// TIA Portal project "TestwithPSC" (V20)

(* hardware
DEVICE "S7-1500/ET200MP station_1"  S7-1500 station
   slot 0: "Rail_0"  Rack  6ES7 590-1***0-0AA0
   slot 1: "PLC_1"  CPU 1516F-3 PN/DP  6ES7 516-3FN01-0AB0  V2.9
      slot 3: "CPU display_1"  6ES7591-1BA00-0AA0
      slot 32768: "PROFINET interface_1"  X1
      slot 33024: "PROFINET interface_2"  X2
      slot 33280: "DP interface_1"  X3
      slot 34817: "Virtual CP interface port_1"  Virtual CP interface port  Virtual CP interface port
DEVICE "GSD device_1"  GSD.Device.PN
   slot 0: "Rack"  Rack  V1.0
   slot 0: "PSC1-C-xxx-FB1-PNPS"  PSC1-C-xxx RE/PNS V3.5.35 - V3.5.x  0000.000  V1.5
      slot 0: "PSC1-C-xxx RE/PNS V3.5.35 - V3.5.x"  PSC1-C-xxx RE/PNS V3.5.35 - V3.5.x
      slot 1: "PN-IO"  PN-IO
         slot 1: "Port 1"  Port 1
         slot 2: "Port 2"  Port 2
   slot 1: "Device Diagnosis_1"  Device Diagnosis
      slot 0: "128 Bytes Input"  128 Bytes Input
   slot 2: "Outputs_1"  Outputs
      slot 0: "4 Bytes Output"  4 Bytes Output
   slot 3: "SD Bus Input_1"  SD Bus Input
      slot 0: "64 Bytes Input"  64 Bytes Input
   slot 4: "SD Bus Output_1"  SD Bus Output
      slot 0: "64 Bytes Output"  64 Bytes Output
   slot 5: "F-Module I/O (12 Bytes)_1"  F-Module I/O (12 Bytes)
      slot 0: "F-Module I/O (12 Bytes)"  F-Module I/O (12 Bytes)
*)

// ===== PLC "PLC_1"  CPU 1516F-3 PN/DP =====

VAR_GLOBAL   // PLC tag table "Default tag table"
   "mReset" AT %M30.0 : Bool;
   "mReset1" AT %M3.1 : Bool;
   "mNetworkResetCmd" AT %M3.2 : Bool;
   "SafetyResetNetworkCmd" AT %Q200.0 : Bool;
   "SafetyINLightCurtain" AT %I200.0 : Bool;
END_VAR

VAR_GLOBAL   // PLC tag table "Tag table_1"
   "PSC1_RawData_IN" AT %I0.0 : "udt_128Bytes";
   "PSC1_RawData_OUT" AT %Q0.0 : "udt_4Bytes";
END_VAR

TYPE "udt_PSC_IN"
   STRUCT
      PSCMode : UInt;
      AliveCounter : UInt;
      DeviceError : UInt;
      ErrorCode : UInt;
      LogicData : Array[0..407] of Bool;
   END_STRUCT;
END_TYPE

TYPE "udt_PSC_OUT"
   STRUCT
      LogicData : Array[0..31] of Bool;
   END_STRUCT;
END_TYPE

TYPE "udt_128Bytes"
   STRUCT
      _raw : Array[0..127] of Byte;
   END_STRUCT;
END_TYPE

TYPE "udt_PSC"
   STRUCT
      in : "udt_PSC_IN";
      out : "udt_PSC_OUT";
   END_STRUCT;
END_TYPE

TYPE "udt_4Bytes"
   STRUCT
      _raw : Array[0..3] of Byte;
   END_STRUCT;
END_TYPE

DATA_BLOCK "Main_Safety_RTG1_DB"   // DB1, F_DB
{ S7_Optimized_Access := 'TRUE' }
NAME : FUSI
VERSION : 0.1
// stored: InstanceOfName Main_Safety_RTG1
"Main_Safety_RTG1"
BEGIN
END_DATA_BLOCK

DATA_BLOCK "FB_PSC_DB"   // DB2
{ S7_Optimized_Access := 'TRUE' }
VERSION : 0.1
// stored: InstanceOfName FB_PSC
"FB_PSC"
BEGIN
END_DATA_BLOCK

DATA_BLOCK "DB_PSC"   // DB3
{ S7_Optimized_Access := 'TRUE' }
VERSION : 0.1
BEGIN
END_DATA_BLOCK

DATA_BLOCK "FB_Station_DB"   // DB4
{ S7_Optimized_Access := 'TRUE' }
VERSION : 0.1
// stored: InstanceOfName FB_Station
"FB_Station"
BEGIN
END_DATA_BLOCK

FUNCTION_BLOCK "Main_Safety_RTG1"   // FB1, F_FBD
{ S7_Optimized_Access := 'TRUE' }
   VAR
      ACK_GL_Instance : ACK_GL;
   END_VAR
   VAR_TEMP
      LightCurtainOK : Bool;
   END_VAR
BEGIN

REGION Network 1
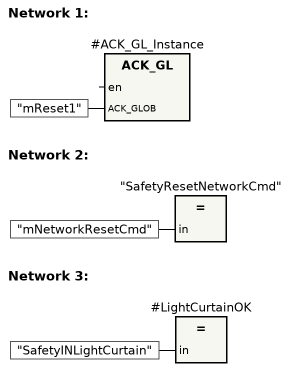
   #ACK_GL_Instance(ACK_GLOB := "mReset1");   // ACK_GL
END_REGION

REGION Network 2
   "SafetyResetNetworkCmd" := "mNetworkResetCmd";
END_REGION

REGION Network 3
   #LightCurtainOK := "SafetyINLightCurtain";
END_REGION
END_FUNCTION_BLOCK

FUNCTION_BLOCK "FB_PSC"   // FB2, LAD
{ S7_Optimized_Access := 'TRUE' }
VERSION : 0.1
   VAR_IN_OUT
      ioRawinputData : Array[*] of Byte;
      ioRawOutputData : Array[*] of Byte;
      ioData : "udt_PSC";
   END_VAR
   VAR_TEMP
      iCounter : Int;
      iIndex : Int;
   END_VAR
BEGIN

REGION Network 2 (SCL)
   #iIndex := 0;
   FOR #iCounter := 5 TO 55 DO

       #ioData.in.LogicData[#iIndex*8]:=
       #ioRawinputData[#iCounter].%X0;

       #ioData.in.LogicData[#iIndex*8+1] :=
       #ioRawinputData[#iCounter].%X1;

       #ioData.in.LogicData[#iIndex*8+2] :=
       #ioRawinputData[#iCounter].%X2;

       #ioData.in.LogicData[#iIndex * 8 + 3] :=
       #ioRawinputData[#iCounter].%X3;

       #ioData.in.LogicData[#iIndex*8+4] :=
       #ioRawinputData[#iCounter].%X4;

       #ioData.in.LogicData[#iIndex * 8 + 5] :=
       #ioRawinputData[#iCounter].%X5;

       #ioData.in.LogicData[#iIndex * 8 + 6] :=
       #ioRawinputData[#iCounter].%X6;

       #ioData.in.LogicData[#iIndex * 8 + 7] :=
       #ioRawinputData[#iCounter].%X7;

       #iIndex := #iIndex + 1;
   END_FOR;
END_REGION

REGION Network 3 (SCL)
   #iIndex := 0;
   FOR #iCounter := 0 TO 3 DO

       #ioRawOutputData[#iCounter].%X0 := #ioData.out.LogicData[#iIndex * 8 + 0];
       #ioRawOutputData[#iCounter].%X1 := #ioData.out.LogicData[#iIndex * 8 + 1];
       #ioRawOutputData[#iCounter].%X2 := #ioData.out.LogicData[#iIndex * 8 + 2];
       #ioRawOutputData[#iCounter].%X3 := #ioData.out.LogicData[#iIndex * 8 + 3];
       #ioRawOutputData[#iCounter].%X4 := #ioData.out.LogicData[#iIndex * 8 + 4];
       #ioRawOutputData[#iCounter].%X5 := #ioData.out.LogicData[#iIndex * 8 + 5];
       #ioRawOutputData[#iCounter].%X6 := #ioData.out.LogicData[#iIndex * 8 + 6];
       #ioRawOutputData[#iCounter].%X7 := #ioData.out.LogicData[#iIndex * 8 + 7];


       #iIndex := #iIndex + 1;
   END_FOR;
END_REGION
END_FUNCTION_BLOCK

FUNCTION_BLOCK "FB_Station"   // FB3, LAD
{ S7_Optimized_Access := 'TRUE' }
VERSION : 0.1
   VAR_INPUT
      iReset : Bool;
   END_VAR
   VAR_OUTPUT
      oLightCurtain : Bool;
      oESTOP : Bool;
      oDoorLockPosition : Bool;
      oDoorOK : Bool;
      oDoorOut1 : Bool;
      oDoorOut2 : Bool;
      oDoorLockUnlock : Bool;
      oEnable : Bool;
   END_VAR
   VAR_IN_OUT
      ioData : "udt_PSC";
   END_VAR
BEGIN

REGION Network 1
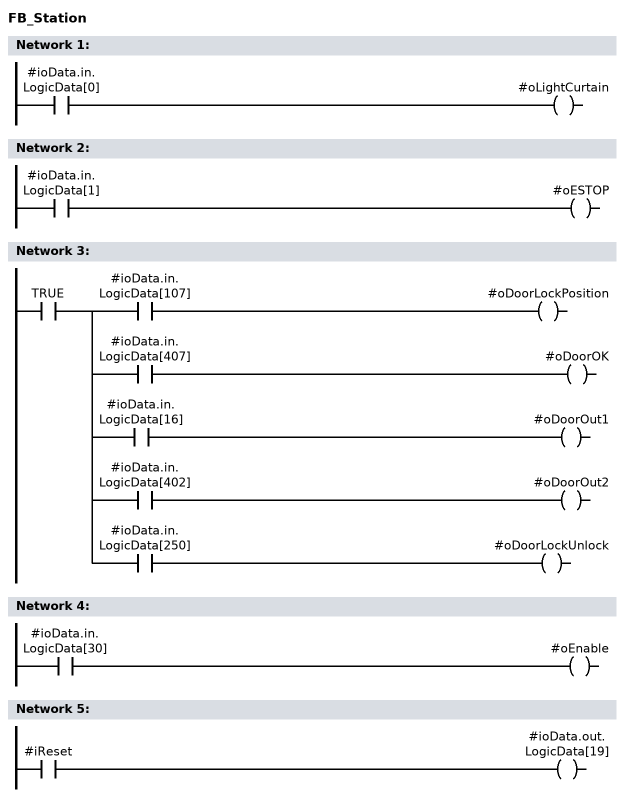
   RUNG wire#powerrail
      Contact( #ioData.in.LogicData[0] )
      Coil( #oLightCurtain )
   END_RUNG
   // the same network as SCL:
   #oLightCurtain := #ioData.in.LogicData[0];
END_REGION

REGION Network 2
   RUNG wire#powerrail
      Contact( #ioData.in.LogicData[1] )
      Coil( #oESTOP )
   END_RUNG
   // the same network as SCL:
   #oESTOP := #ioData.in.LogicData[1];
END_REGION

REGION Network 3
   RUNG wire#powerrail
      Contact( TRUE )
      wire#w1
      Contact( #ioData.in.LogicData[107] )
      Coil( #oDoorLockPosition )
   END_RUNG
   RUNG wire#w1
      Contact( #ioData.in.LogicData[407] )
      Coil( #oDoorOK )
   END_RUNG
   RUNG wire#w1
      Contact( #ioData.in.LogicData[16] )
      Coil( #oDoorOut1 )
   END_RUNG
   RUNG wire#w1
      Contact( #ioData.in.LogicData[402] )
      Coil( #oDoorOut2 )
   END_RUNG
   RUNG wire#w1
      Contact( #ioData.in.LogicData[250] )
      Coil( #oDoorLockUnlock )
   END_RUNG
   // the same network as SCL:
   #oDoorLockPosition := TRUE AND #ioData.in.LogicData[107];
   #oDoorOK := TRUE AND #ioData.in.LogicData[407];
   #oDoorOut1 := TRUE AND #ioData.in.LogicData[16];
   #oDoorOut2 := TRUE AND #ioData.in.LogicData[402];
   #oDoorLockUnlock := TRUE AND #ioData.in.LogicData[250];
END_REGION

REGION Network 4
   RUNG wire#powerrail
      Contact( #ioData.in.LogicData[30] )
      Coil( #oEnable )
   END_RUNG
   // the same network as SCL:
   #oEnable := #ioData.in.LogicData[30];
END_REGION

REGION Network 5
   RUNG wire#powerrail
      Contact( #iReset )
      Coil( #ioData.out.LogicData[19] )
   END_RUNG
   // the same network as SCL:
   #ioData.out.LogicData[19] := #iReset;
END_REGION
END_FUNCTION_BLOCK

ORGANIZATION_BLOCK "Main"   // OB1, LAD, ProgramCycle
TITLE = "Main Program Sweep (Cycle)"
{ S7_Optimized_Access := 'TRUE' }
VERSION : 0.1
   VAR_INPUT
      Initial_Call : Bool;   // Initial call of this OB
      Remanence : Bool;   // =True, if remanent data are available
   END_VAR
   VAR_TEMP   // added for the SCL form of the ladder/FBD networks
      _w1 : Bool;
   END_VAR
BEGIN

REGION Network 2
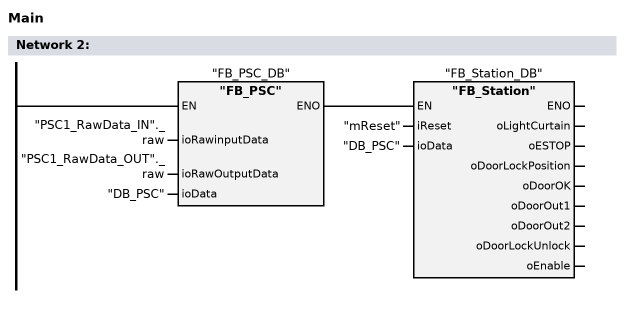
   RUNG wire#powerrail
      "FB_PSC_DB"(ioRawinputData := "PSC1_RawData_IN"._raw, ioRawOutputData := "PSC1_RawData_OUT"._raw, ioData := "DB_PSC")
      "FB_Station_DB"(iReset := "mReset", ioData := "DB_PSC", oLightCurtain =>, oESTOP =>, oDoorLockPosition =>, oDoorOK =>, oDoorOut1 =>, oDoorOut2 =>, oDoorLockUnlock =>, oEnable =>)
   END_RUNG
   // the same network as SCL:
   "FB_PSC_DB"(ioRawinputData := "PSC1_RawData_IN"._raw,   // "FB_PSC"
               ioRawOutputData := "PSC1_RawData_OUT"._raw,
               ioData := "DB_PSC",
               ENO => #_w1);
   IF #_w1 THEN
       "FB_Station_DB"(iReset := "mReset", ioData := "DB_PSC");   // "FB_Station"
   END_IF;
END_REGION
END_ORGANIZATION_BLOCK